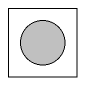
[picture p262: PARTRESULT (HMI screen)]
ellipse at (12,12)-(57,57): invisible if ($PartResult$ MOD 10) = 0; alarm colour if ($PartResult$ MOD 10) <> 1
ellipse at (12,12)-(57,57): invisible if ($PartResult$ MOD 10) <> 4
ellipse at (12,12)-(57,57): invisible if ($PartResult$ MOD 10) <> 5
ellipse at (12,12)-(57,57): invisible if ($PartResult$ MOD 10) <> 0
1 more shapes without text or variables
*)
